TYPE DUT_State_Motor_Freq_Enum : (
    Off := 0,
	Starting := 10,
	On := 20,
	Stopping := 30
);
END_TYPE

(* stored: Version 1.1.0.1, ProductVersion 3.1.4024.12
   DUT DUT_State_Motor_Freq_Enum: Id {3646c610-fd56-4c8a-a496-166f7156fd0f} *)
